// TIA Portal project "ProfiEcho" (V17)

(* hardware
DEVICE "S7-1500/ET200MP-Station_1"  S7-1500 station
   slot 0: "Profilschiene_0"  Rack  6ES7 590-1***0-0AA0
   slot 1: "PLC_1"  CPU 1516-3 PN/DP  6ES7 516-3AN01-0AB0  V2.9
      slot 3: "CPU-Display_1"  6ES7591-1BA00-0AA0
      slot 32768: "PROFINET-Schnittstelle_1"  X1
      slot 33024: "PROFINET-Schnittstelle_2"  X2
      slot 33280: "DP-Schnittstelle_1"  X3
      slot 34817: "Virtual CP interface port_1"  Virtual CP interface port  Virtual CP interface port
DEVICE "GSD-Geraet_1"  GSD.Device.PN
   slot 0: "Baugruppenträger"  Rack  V1.0
   slot 0: "profiecho"  Profiecho  123 444 555  V0.1.0
      slot 0: "Profiecho"  Profiecho
      slot 1: "X1"  X1
         slot 1: "X1 P1"  X1 P1
      slot 1: "unknown module_1"  unknown module  1.0
         slot 0: "unknown submodule"  unknown submodule
*)

// ===== PLC "PLC_1"  CPU 1516-3 PN/DP =====

VAR_GLOBAL   // PLC tag table "Standard-Variablentabelle"
   "EchoFloatIn" AT %ID0 : Real;
   "EchoIntIn" AT %ID4 : UDInt;
   "EchoFloatOut" AT %QD0 : Real;
   "EchoIntOut" AT %QD4 : UDInt;
   "Tag_1" AT %M0.0 : Bool;
END_VAR

// folder: System blocks/Program resources

DATA_BLOCK "IEC_Timer_0_DB"   // DB1
{ S7_Optimized_Access := 'TRUE' }
AUTHOR : Simatic
FAMILY : IEC
NAME : IEC_TMR
VERSION : 1.0
// stored: InstanceOfName IEC_TIMER
"IEC_TIMER"
BEGIN
END_DATA_BLOCK

DATA_BLOCK "IEC_Timer_0_DB_1"   // DB2
{ S7_Optimized_Access := 'TRUE' }
AUTHOR : Simatic
FAMILY : IEC
NAME : IEC_TMR
VERSION : 1.0
// stored: InstanceOfName IEC_TIMER
"IEC_TIMER"
BEGIN
END_DATA_BLOCK

// folder: (top level)

ORGANIZATION_BLOCK "Main"   // OB1, LAD, ProgramCycle
TITLE = "Main Program Sweep (Cycle)"
{ S7_Optimized_Access := 'TRUE' }
VERSION : 0.1
   VAR_INPUT
      Initial_Call : Bool;   // Initial call of this OB
      Remanence : Bool;   // =True, if remanent data are available
   END_VAR
   VAR_TEMP
      tempFloatIn : Real;
      tempIntIn : UDInt;
      tempFloatOut : Real;
   END_VAR
BEGIN

REGION Network 1
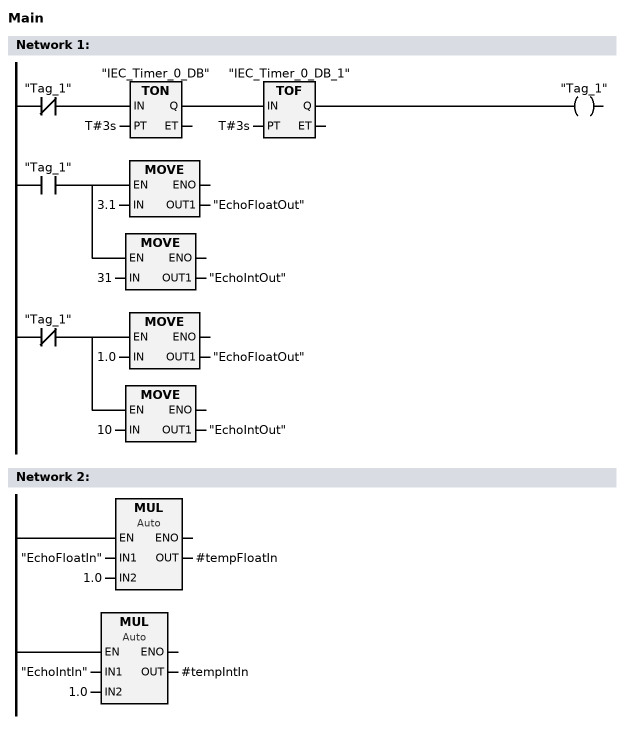
   "IEC_Timer_0_DB".TON(IN := NOT "Tag_1", PT := T#3s);
   "IEC_Timer_0_DB_1".TOF(IN := "IEC_Timer_0_DB".Q, PT := T#3s);
   "Tag_1" := "IEC_Timer_0_DB_1".Q;
   IF "Tag_1" THEN
       "EchoFloatOut" := 3.1;
       "EchoIntOut" := 31;
   END_IF;
   IF NOT "Tag_1" THEN
       "EchoFloatOut" := 1.0;
       "EchoIntOut" := 10;
   END_IF;
END_REGION

REGION Network 2
   RUNG wire#powerrail
      Mul(in1 := "EchoFloatIn", in2 := 1.0, out => #tempFloatIn)
   END_RUNG
   RUNG wire#powerrail
      Mul(in1 := "EchoIntIn", in2 := 1.0, out => #tempIntIn)
   END_RUNG
   // the same network as SCL:
   #tempFloatIn := "EchoFloatIn" * 1.0;
   #tempIntIn := "EchoIntIn" * 1.0;
END_REGION
END_ORGANIZATION_BLOCK